RoboDK station: UR3E_Station_Red_Yellow_Classify.rdk

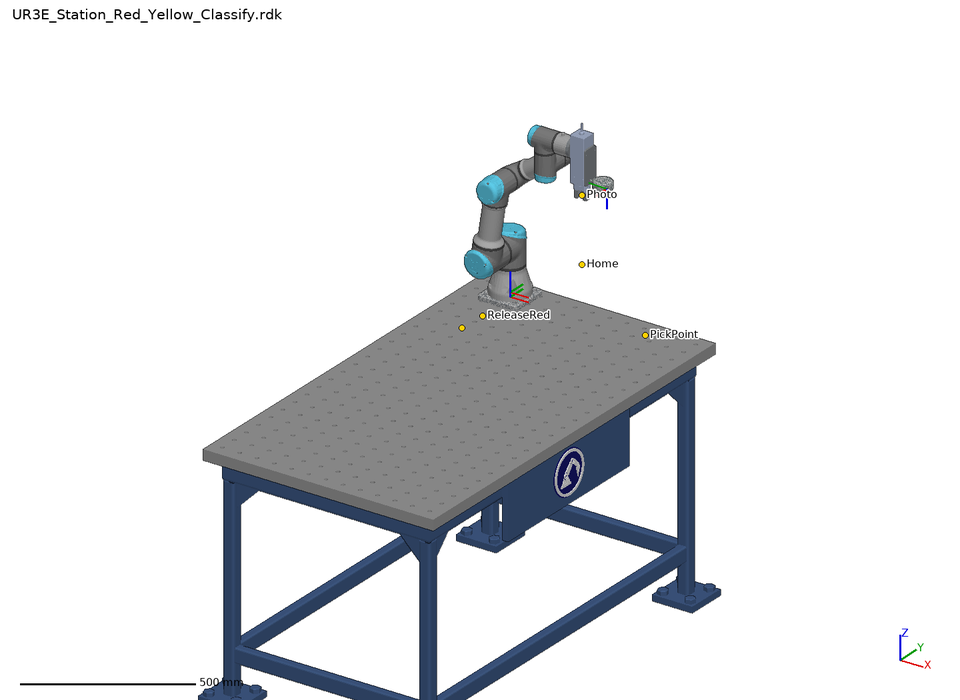
[picture v0: the station drawn from its stored meshes, robots at their saved joint values, targets as dots, program paths as lines]
Station UR3E_Station_Red_Yellow_Classify (saved by RoboDK 5.2.5). Poses are relative to the parent item; angles as X-Y-Z fixed-axis rotations.
Station parameters (name, value as stored): IO_5, 1, IO_10, 0, RECORD_READY, 0, True, 0, IO_11, 0
  - frame World Frame at (0, 0, 0) mm
    - frame UR3e Base at (0, 0, 15) mm
      - robot UR3e: 6 axes, payload 3 kg, reach 500 mm, repeatability 0.03 mm, weight 11 kg
          modified DH rows (alpha deg, a mm, theta deg, d mm): 0, 0, 0, 151.9; 90, 0, 180, 0; 0, 243.55, 0, 0; 0, 213.2, 0, 131.05; -90, 0, 0, 85.35; 90, 0, 180, 92.1
          joint limits [-360, -360, -360, -360, -360, -360] to [360, 360, 360, 360, 360, 360]; home [0, -90, -90, 0, 90, 0]; saved at [-0.002, -98.741, -47.006, -34.261, 89.995, 0]
        - tool Gripper, TCP at (0, 145, 35) mm, size 63 x 236.5 x 138.7 mm, geometry from RGI14_cBrida_UR3e.STEP
        - frame Camera Frame at (-1.25, 99.12, 122.31) mm, rotated rx -89.49 ry 0.51 rz -0.14 deg
          - camera My Camera
      - target PickPoint (Cartesian target) at (484.35, -21.86, 7.24) mm, rotated rx -90 ry 0 rz -90 deg; joints [17.976, -156.363, -82.591, 58.953, 72.022, 0.001] of UR3e
      - target Photo (Cartesian target) at (340.3, -131.05, 453) mm, rotated rx -90 ry 0 rz -90 deg; joints [0, -100.092, -43.022, -36.886, 90, 0] of UR3e
    - object Table 1400x800x800mm at (250, -250, 0) mm, rotated rx 0 ry 0 rz -90 deg, size 1420 x 820 x 800 mm, geometry from Table-1400x800x800mm.sld
    - object Mounting_Plate_UR3e at (0, 0, 0) mm, size 140 x 140 x 15 mm, geometry from Mounting_Plate_UR3e.stp
    - target Home (Cartesian target) at (340.3, -131.05, 250) mm, rotated rx -90 ry 0 rz -90 deg; joints [0, -95.015, -110.808, 25.823, 90, 0] of UR3e
    - target ReleaseRed (Cartesian target) at (136.05, -329.9, 108.92) mm, rotated rx -90.2 ry -0.28 rz 177.77 deg; joints [-23.235, -122.01, -125.79, 67.229, 21.005, 0.249] of UR3e
    - target ReleaseYellow (Cartesian target) at (135.8, -431.39, 110.89) mm, rotated rx -90.21 ry -0.25 rz 177.81 deg; joints [-42.192, -134.564, -95.056, 49.287, 40.003, 0.003] of UR3e
  - program Home_Position (4 instructions, listed below)
  - program Pick_Position (3 instructions, listed below)
  - program Gripper Open (2 instructions, listed below)
  - program Gripper Close (2 instructions, listed below)
  - program Gripper_TurnH (2 instructions, listed below)
  - program Gripper_TurnV (2 instructions, listed below)
  - program Image Capture Position (3 instructions, listed below)
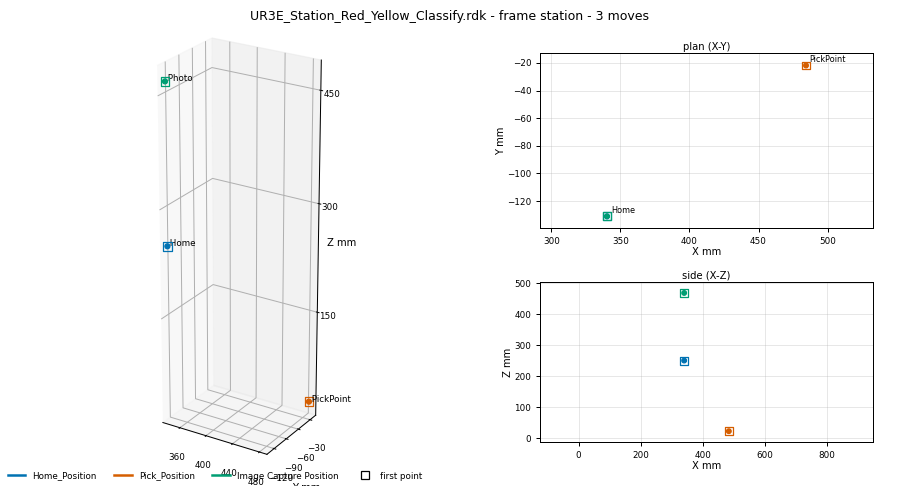
[picture p0: tool path of UR3E_Station_Red_Yellow_Classify.rdk in frame station, 3 of 3 moves have a stored position in this frame; points joined in program order, loops and branches not executed]

--- program Home_Position (robot UR3e) ---
  Set Ref.: World Frame
  Set Tool: Gripper
  MoveJ (Home)
  Set speed (50.0 deg/s)

--- program Pick_Position (robot UR3e) ---
  Set Ref.: World Frame
  Set Tool: Gripper
  MoveJ (PickPoint)

--- program Gripper Open (robot UR3e) ---
  Set IO_10=1
  Pause 500 ms

--- program Gripper Close (robot UR3e) ---
  Set IO_10=0
  Pause 500 ms

--- program Gripper_TurnH (robot UR3e) ---
  Set IO_11=1
  Pause 500 ms

--- program Gripper_TurnV (robot UR3e) ---
  Set IO_11=0
  Pause 500 ms

--- program Image Capture Position (robot UR3e) ---
  Set Ref.: UR3e Base
  Set Tool: Gripper
  MoveJ (Photo)
